PROGRAM P30_GasFlowControl
VAR
	//bMaxValueChanged : BOOL;
	aMFC : ARRAY[1..19] OF FB_RampGeneration_Gas; //MFC 0 ~ 5V
	aEPC : ARRAY[1..7] OF FB_RampGeneration_Gas; //EPC 0 ~ 5V
	aMFC_TV : ARRAY[1..19] OF INT;
	aMFC_RampTime : ARRAY[1..19] OF INT;
	aMFC_PV : ARRAY[1..19] OF INT;
	aEPC_TV : ARRAY[1..7] OF INT;
	aEPC_RampTime : ARRAY[1..7] OF INT;
	aEPC_PV	: ARRAY[1..7] OF INT;
	i 	: INT;
	j 	: INT;
END_VAR

VAR CONSTANT
	KL3464MaxValueH	: REAL := 16383; //0~5V Half Input
	//KL4404MaxValueH	: REAL := 16383; //0~5V Half Output
END_VAR

//Tempeary Value for TEST
GVL_IO.aMaxValue[1] := 4000; //MFC1 MO Manifold RUN
GVL_IO.aMaxValue[2] := 4000; //MFC2 HYD Manifold RUN
GVL_IO.aMaxValue[3] := 4000; //MFC3 NH3 #1
GVL_IO.aMaxValue[4] := 4000; //MFC4 NH3 #2
GVL_IO.aMaxValue[8] := 50; //MFC4 NH3 #2
GVL_IO.aMaxValue[20] := 2000; //EPC
GVL_IO.aMaxValue[21] := 2250; //EPC
GVL_IO.aMaxValue[22] := 2250; //EPC
GVL_IO.aMaxValue[23] := 2250; //EPC
GVL_IO.aMaxValue[24] := 2250; //EPC
GVL_IO.aMaxValue[25] := 2250; //EPC
GVL_IO.aMaxValue[26] := 2250; //EPC
//aMFC_RampTime[i]; <-- Frome UI
//aMFC_TV[i] <-- From UI

//IF bMaxValueChanged THEN
//	FOR i:=1 TO 4 DO
//		aMFC[i].rMaxValue := GVL_IO.aMaxValue[i];
//	END_FOR								
//END_IF

(* Read from Device*)
FOR i:=1 TO 19 DO
	IF GVL_IO.aMaxValue[i] <> 0 THEN
		aMFC[i].nState := 1;
		aMFC[i].nRampTime := aMFC_RampTime[i];
		aMFC[i].rTargetValue := aMFC_TV[i] / GVL_IO.aMaxValue[i] * KL3464MaxValueH; //Input Set Value
		GVL_IO.aAnalogOutputIO[i] := LREAL_TO_INT(aMFC[i].rControlValue);
		
		aMFC_PV[i] := REAL_TO_INT(GVL_IO.aAnalogInputIO[i] / KL3464MaxValueH * GVL_IO.aMaxValue[i]);
		aMFC[i]();
	END_IF
END_FOR

FOR i:=1 TO 7 DO
	j := i + 19; //Offset Analog Input Output Card
	IF GVL_IO.aMaxValue[j] <> 0 THEN
		aEPC[i].nState := 1;
		aEPC[i].nRampTime := aEPC_RampTime[i];
		aEPC[i].rTargetValue := aEPC_TV[i] / GVL_IO.aMaxValue[j] * KL3464MaxValueH; //Input Set Value
		GVL_IO.aAnalogOutputIO[j] := LREAL_TO_INT(aEPC[i].rControlValue);
		
		aEPC_PV[i] := REAL_TO_INT(GVL_IO.aAnalogInputIO[j] / KL3464MaxValueH * GVL_IO.aMaxValue[j]);
		
		aEPC[i]();
	END_IF
END_FOR

END_PROGRAM

(* stored: Version 1.1.0.1, ProductVersion 3.1.4026.8
   POU P30_GasFlowControl: Id {761008bd-d9bc-489c-85ce-c898e802d93f}, SpecialFunc None *)
